TYPE EL6xxx22ByteOutData :
STRUCT
	Control : WORD;     
	Data : ARRAY [0..21] OF BYTE; 
END_STRUCT
END_TYPE

(* stored: Version 1.1.0.1, ProductVersion 3.1.4026.18
   DUT EL6xxx22ByteOutData: Id {f27cbe5d-3ead-4d18-a3ef-8fe69f6f0b05} *)
